# EPICS substitutions: db/core/ecmcEcTiming.substitutions
file "ecmcEcTiming.template"
{
  pattern { DIR_PV, DIR_ASYN }
          { "In",   "input"  }
          { "Out",  "output" }
}
